Staubli VAL3: SparePoint.dtx

bool bByPass[4]
bool bExit
bool bListRefresh
bool bUserRefresh
frame fFrame = {fatherId=world[0]}
mdesc mNomSpeed
num nPage = 1
num nSelected
public pointRx pPoint{}
  [P1] = {x=495.660657, y=122.165524, z=84.338304, rx=9.53283, ry=179.762496, rz=-66.438432, shoulder=lefty, elbow=epositive, wrist=wpositive, fatherId=world[0]}
  [P10] = {fatherId=world[0]}
  [P11] = {fatherId=world[0]}
  [P12] = {fatherId=world[0]}
  [P13] = {fatherId=world[0]}
  [P14] = {fatherId=world[0]}
  [P15] = {fatherId=world[0]}
  [P16] = {fatherId=world[0]}
  [P2] = {fatherId=world[0]}
  [P3] = {fatherId=world[0]}
  [P4] = {fatherId=world[0]}
  [P5] = {fatherId=world[0]}
  [P6] = {fatherId=world[0]}
  [P7] = {fatherId=world[0]}
  [P8] = {fatherId=world[0]}
  [P9] = {fatherId=world[0]}
public string sDeli[2]
  [0] = "A"
  [1] = "C"
public string sFileList = "A140"
string sFolder = "Disk://Traj/"
string sItem = "P1"
string sList[16]
  [0] = "P1"
  [1] = "P2"
  [2] = "P3"
  [3] = "P4"
  [4] = "P5"
  [5] = "P6"
  [6] = "P7"
  [7] = "P8"
  [8] = "P9"
  [9] = "P10"
  [10] = "P11"
  [11] = "P12"
  [12] = "P13"
  [13] = "P14"
  [14] = "P15"
  [15] = "P16"
string sListItemValue
string sOutputFolder = "Disk://Traj/"
string sParameter
string sPointName = "P1"
string sPtPara
